(* IEC 61131-3 sources: CodesysTest/alpha/export/PAM.dev/Plc Logic/Application/Motors/Applied Motion/DataHandlers/FB_StepServoCommands.pou/FeedToPosition.prop, 1 file *)

(* ---- Set.pm.st ---- *)
(*#-#-#-#-#-#-#-#-#-#---Declaration---#-#-#-#-#-#-#-#-#-#-#-#-#*)

VAR
END_VAR
(*#-#-#-#-#-#-#-#-#-#---Implementation---#-#-#-#-#-#-#-#-#-#-#-#-#*)

commandSent := FALSE;
_feedToPosition := FeedToPosition;
